SUBAPPLICATION Uebung_039_sub_NumbAnzeig (* Subapplication Type *)
  (* Standard: 61499-2 *)
  (* Version 1.0, 2024-03-03, franz *)
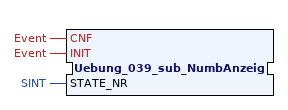
  EVENT_INPUT
    CNF;
    INIT;
  END_EVENT
  VAR_INPUT
    STATE_NR : SINT;
  END_VAR
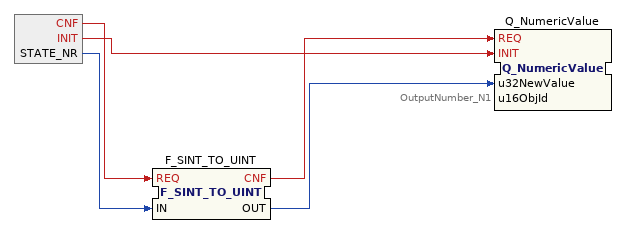
  FBS
    F_SINT_TO_UINT : F_SINT_TO_UINT;
    Q_NumericValue : Q_NumericValue(u16ObjId := OutputNumber_N1);
  END_FBS
  EVENT_CONNECTIONS
    F_SINT_TO_UINT.CNF TO Q_NumericValue.REQ;
    CNF TO F_SINT_TO_UINT.REQ;
    INIT TO Q_NumericValue.INIT;
  END_CONNECTIONS
  DATA_CONNECTIONS
    F_SINT_TO_UINT.OUT TO Q_NumericValue.u32NewValue;
    STATE_NR TO F_SINT_TO_UINT.IN;
  END_CONNECTIONS
END_SUBAPPLICATION
